(* PLC project cp_door, Dassault Systèmes ControlBuild 2024x *)
(* stored: creationDateTime 2023-10-03T11:13:50-01:00 *)

FUNCTION_BLOCK tni_train.cp_door
  VAR_INPUT
    enableOpening : BOOL := false;
    enableClosing : BOOL := false;
  END_VAR
  VAR_INPUT
    openedDoor : BOOL := false;
    closedDoor : BOOL := false;
  END_VAR
  VAR_INPUT
    lockedDoor : BOOL := false;
    unlockedDoor : BOOL := false;
  END_VAR
  VAR_INPUT
    openingRequest : BOOL := false;
  END_VAR
  VAR_OUTPUT
    doorOpeningCmd : BOOL := false;
    doorClosingCmd : BOOL := false;
  END_VAR
  VAR_OUTPUT
    doorLockingCmd : BOOL := false;
    doorUnlockingCmd : BOOL := false;
  END_VAR
  VAR_OUTPUT
    closedDoorState : BOOL := false;
    openedDoorState : BOOL := false;
    faultState : DINT := 0;
  END_VAR

INITIAL_STEP 10:
  10_INLINE1(N);
  COMPUTE_FUNCTION_BLOCKS(S);
END_STEP
ACTION 10_INLINE1:
  closedDoorState;
END_ACTION
TRANSITION FROM 10 TO 11
  := enableOpening;
END_TRANSITION
STEP 11:
  11_INLINE2(N);
END_STEP
ACTION 11_INLINE2:
  doorUnlockingCmd;
END_ACTION
TRANSITION FROM 11 TO 12
  := unlockedDoor;
END_TRANSITION
STEP 12:
END_STEP
TRANSITION FROM 12 TO 13
  := openingRequest;
END_TRANSITION
TRANSITION FROM 12 TO 16
  := NOT enableOpening;
END_TRANSITION
STEP 13:
  13_INLINE3(N);
END_STEP
ACTION 13_INLINE3:
  doorOpeningCmd;
END_ACTION
TRANSITION FROM 13 TO 14
  := openedDoor;
END_TRANSITION
STEP 14:
  14_INLINE4(N);
END_STEP
ACTION 14_INLINE4:
  openedDoorState;
END_ACTION
TRANSITION FROM 14 TO 15
  := enableClosing;
END_TRANSITION
STEP 15:
  15_INLINE5(N);
END_STEP
ACTION 15_INLINE5:
  doorClosingCmd;
END_ACTION
TRANSITION FROM 15 TO 16
  := closedDoor;
END_TRANSITION
STEP 16:
  16_INLINE6(N);
END_STEP
ACTION 16_INLINE6:
  doorLockingCmd;
END_ACTION
TRANSITION FROM 16 TO 10
  := lockedDoor;
END_TRANSITION
ACTION COMPUTE_FUNCTION_BLOCKS:  (* blocks drawn on the SFC sheet *)
  G1:
END_ACTION
END_FUNCTION_BLOCK
